SYSTEM PackageRenameTest
  (* Version 1.0, 2026-07-29, Dimitrios Kalligaridis *)
  APPLICATION App
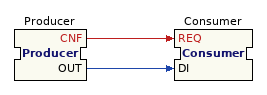
    FBS
      Producer : mypackage::Producer;
      Consumer : mypackage::Consumer;
    END_FBS
    EVENT_CONNECTIONS
      Producer.CNF TO Consumer.REQ;
    END_CONNECTIONS
    DATA_CONNECTIONS
      Producer.OUT TO Consumer.DI;
    END_CONNECTIONS
  END_APPLICATION
END_SYSTEM
